// TIA Portal V16 export
// export: Created 2023-03-29T11:03:47.2302545Z, ExportSetting WithDefaults, DisplayName Totally Integrated Automation Portal, DisplayVersion V16 Update 6, DisplayName TIA Portal Version Control Interface, DisplayVersion V16 Update 2, DisplayName TIA Portal Openness, DisplayVersion V16 Update 6, DisplayName STEP 7 Professional, DisplayVersion V16 Update 6, DisplayName STEP 7 Safety, DisplayVersion V16, DisplayName WinCC Advanced, DisplayVersion V16 Update 6
VAR_GLOBAL   // PLC tag table "zbiorniki"
   set_HWork_Tank_3 AT %M45.2 : Bool;   // bit statusu aktywacji zbiornika do pracy w trybie sekwencji
   set_HWork_Tank_1 AT %M45.0 : Bool;   // bit statusu aktywacji zbiornika do pracy w trybie sekwencji
   set_HWork_Tank_2 AT %M45.1 : Bool;   // bit statusu aktywacji zbiornika do pracy w trybie sekwencji
   set_HWork_Tank_4 AT %M45.3 : Bool;   // bit statusu aktywacji zbiornika do pracy w trybie sekwencji
   mem_set_auto_zb_3 AT %M82.2 : Bool;   // ustawione w sekwencji jako aktywna
   blok_tank_3 AT %M82.6 : Bool;   // jest zablokowany po pracy w sekwencji
   blok_tank_1 AT %M82.4 : Bool;   // jest zablokowany po pracy w sekwencji
   mem_set_auto_zb_2 AT %M82.1 : Bool;   // ustawione w sekwencji jako aktywna
   blok_tank_4 AT %M82.7 : Bool;   // jest zablokowany po pracy w sekwencji
   act_Eptying AT %M45.4 : Bool;   // trwa procedura pompowania
   mem_set_auto_zb_1 AT %M82.0 : Bool;   // ustawione w sekwencji jako aktywna
   memTrig_set_manual_zb_4 AT %M83.3 : Bool;   // ustaw w automat zasuwę aktywnego zbiornika
   memTrig_set_manual_zb_3 AT %M83.2 : Bool;   // ustaw w automat zasuwę aktywnego zbiornika
   memTrig_set_manual_zb_1 AT %M83.0 : Bool;   // ustaw w automat zasuwę aktywnego zbiornika
   blok_tank_2 AT %M82.5 : Bool;   // jest zablokowany po pracy w sekwencji
   act_Filling AT %M45.5 : Bool;   // trwa procedura napełniania
   mem_set_auto_zb_4 AT %M82.3 : Bool;   // ustawione w sekwencji jako aktywna
   memTrig_set_manual_zb_2 AT %M83.1 : Bool;   // ustaw w automat zasuwę aktywnego zbiornika
END_VAR
